TEXTLIST tlEthercatState
  1 = 'Init'
  2 = 'PreOp'
  3 = 'BootStrap'
  4 = 'SafeOp'
  8 = 'Op'
  10 = 'Error'
  20 = 'InvalidVprs'
  40 = 'InitCmndErr'
  80 = 'Disabled'
   = ''
END_TEXTLIST

(* stored: Version 1.1.0.1, ProductVersion 3.1.4024.12
   TextList tlEthercatState: Id {1434d00c-de39-07f8-139a-89e652273800} *)
